{attribute 'linkalways'} 
{attribute 'no_explicit_call' := 'This FB is a CLASS and must be accessed using methods or properties'}
{attribute 'enable_dynamic_creation'}
FUNCTION_BLOCK _GEV_CAMERA_STATE EXTENDS EnumDatatypeBase
VAR
	localData : GEV_CAMERA_STATE;
	activeData : REFERENCE TO GEV_CAMERA_STATE;
	enumBaseDatatype : _BYTE(localData);
END_VAR

METHOD PRIVATE AddLocalEnumeration
VAR_INPUT
	Enumeration : T_MAXSTRING;
	Value : GEV_CAMERA_STATE;
END_VAR
AddEnumeration(Enumeration, Value);
END_METHOD

PROPERTY PUBLIC Address : PVOID
GET
Address := ADR(activeData);
END_GET
END_PROPERTY

METHOD PUBLIC ClearReference
VAR_INPUT
END_VAR
activeData REF= localData;
SetBaseDatatypeReference();
END_METHOD

METHOD PUBLIC Clone : I_Datatype
VAR
    pClone : POINTER TO _GEV_CAMERA_STATE;
END_VAR
pClone := __NEW(_GEV_CAMERA_STATE(InitialValue := Value));
Clone := pClone^;
END_METHOD

METHOD FB_init : BOOL
VAR_INPUT
	bInitRetains : BOOL; // if TRUE, the retain variables are initialized (warm start / cold start)
	bInCopyCode : BOOL;  // if TRUE, the instance afterwards gets moved into the copy code (online change)
	InitialValue : GEV_CAMERA_STATE;
END_VAR
localData := InitialValue;
AddBaseDatatype(enumBaseDatatype);
ClearReference();

AddLocalEnumeration('GEV_CAMERA_IDLE', GEV_CAMERA_STATE.GEV_CAMERA_IDLE);
AddLocalEnumeration('GEV_CONTROL_CHANNEL_OPEN_MASK', GEV_CAMERA_STATE.GEV_CONTROL_CHANNEL_OPEN_MASK);
AddLocalEnumeration('GEV_STREAM_CHANNELS_OPEN_MASK', GEV_CAMERA_STATE.GEV_STREAM_CHANNELS_OPEN_MASK);
AddLocalEnumeration('GEV_CONTROL_CHANNEL_OPEN', GEV_CAMERA_STATE.GEV_CONTROL_CHANNEL_OPEN);
AddLocalEnumeration('GEV_STREAM_CHANNELS_OPEN', GEV_CAMERA_STATE.GEV_STREAM_CHANNELS_OPEN);
END_METHOD

PROPERTY PUBLIC Identifier : T_MAXSTRING
GET
Identifier := 'GEV_CAMERA_STATE';
END_GET
END_PROPERTY

METHOD IsEnumeratorValueEqual : BOOL
VAR_INPUT
	Enumerator : I_KeyValueForwardEnumerator;
END_VAR
VAR
	storedValue : GEV_CAMERA_STATE;
END_VAR
IF NOT Enumerator.TryGet(storedValue) THEN
	RETURN;
END_IF

IsEnumeratorValueEqual := storedValue = activeData;
END_METHOD

METHOD PUBLIC MakeReferenceTo
VAR_INPUT
	ReferenceTarget : REFERENCE TO GEV_CAMERA_STATE;
END_VAR
activeData REF= ReferenceTarget;
SetBaseDatatypeReference();
END_METHOD

METHOD PROTECTED SetBaseDatatypeReference
VAR_INPUT
END_VAR
enumBaseDatatype.MakeReferenceTo(activeData);
END_METHOD

PROPERTY PUBLIC Size : UDINT
GET
Size := SIZEOF(activeData);
END_GET
END_PROPERTY

METHOD TryMakeReferenceTo : BOOL
VAR_INPUT
	Target : I_Datatype;
END_VAR
VAR
	pTargetData : POINTER TO GEV_CAMERA_STATE;
END_VAR
IF NOT IsEquivalentTo(Target) THEN
	RETURN;
END_IF

pTargetData := Target.Address;
activeData REF= pTargetData^;
SetBaseDatatypeReference();
TryMakeReferenceTo := TRUE;
END_METHOD

PROPERTY PUBLIC Value : GEV_CAMERA_STATE
GET
Value := activeData;
END_GET
SET
activeData := Value;
END_SET
END_PROPERTY

END_FUNCTION_BLOCK

(* stored: Version 1.1.0.1, ProductVersion 3.1.4024.13
   POU _GEV_CAMERA_STATE: Id {52fdcd4b-6506-0b2d-1d7d-a99e4f93d5f5}, SpecialFunc None
   Folder Core: Id {243f790b-9eb7-0b65-1820-4362d36b127f}
   Folder Protected: Id {a3054ec1-097b-0c19-2caa-66ed7d579b8d}
   Folder Customize: Id {53ffcbf3-8221-06f0-2ee7-881a6e055832}
   Folder Constructor: Id {7c449b24-9480-0550-155f-ced8adcf0179}
   Folder Private: Id {5f935d4a-2521-067f-26a6-9e6c4ae6d9e8}
   Folder Protected: Id {32fb7fde-8df9-05d1-1060-86eaeddaf911}
   Method AddLocalEnumeration: Id {3e43ae4c-e992-0125-1867-4ac14cc75cea}
   Property Address: Id {8680c0b3-755d-0132-1f08-51abcf5662b2}
   Get Get: Id {c157cf7e-5b2e-0652-35ea-ceb4a7393dc8}
   Method ClearReference: Id {27b3f09e-2a60-0f16-14cb-3d848b71d07a}
   Method Clone: Id {bb877194-70e1-039b-057e-18ca08f5ff89}
   Method FB_init: Id {77b83ecc-f577-0396-1034-795397f92968}
   Property Identifier: Id {579eebd0-2e37-055d-24b0-09f2199784aa}
   Get Get: Id {ed1e10fa-fc6a-02d5-2a68-df5c8370b6e0}
   Method IsEnumeratorValueEqual: Id {2ec705f5-59e6-0a61-1234-16b59d9bdfe4}
   Method MakeReferenceTo: Id {2d506990-ca5e-01f7-35ff-3a7cdb14eafb}
   Method SetBaseDatatypeReference: Id {61cb3714-eca0-0b18-32e7-8612464c0592}
   Property Size: Id {ef56890f-3c6e-0c88-2463-b44579184b7f}
   Get Get: Id {695a1614-5c4b-08d9-1d49-ce5485276e04}
   Method TryMakeReferenceTo: Id {6fa995f2-77ed-060f-039d-39c5cbd32a45}
   Property Value: Id {b096293c-e353-0c4e-2373-fa2e71dc6e1b}
   Get Get: Id {9a4d8600-a17c-06a6-006f-f4b631578642}
   Set Set: Id {65434d82-9e28-0b27-3d30-56cbce2a2629} *)
